// TIA Portal project "Örnek Asansör" (V16)

(* hardware
DEVICE "S71500/ET200MP station_1"  S7-1500 station
   slot 0: "Rail_0"  Rack  6ES7 590-1***0-0AA0
   slot 1: "PLC_1"  CPU 1517-3 PN/DP  6ES7 517-3AP00-0AB0  V2.8
      slot 3: "CPU display_1"  6ES7591-1BA00-0AA0
      slot 32768: "PROFINET interface_1"  X1
         slot 32769: "Port_1"  X1 P1
         slot 32770: "Port_2"  X1 P2
      slot 33024: "PROFINET interface_2"  X2
         slot 33025: "Port_1"  X2 P1
      slot 33280: "DP interface_1"  X3
      slot 34817: "Virtual CP interface port_1"  Virtual CP interface port  Virtual CP interface port
DEVICE "HMI_1"  TP1500 Comfort
   slot 0: "HMI_1"  TP1500 Comfort  6AV2 124-0QC02-0AX1  16.0.0.0
   slot 1: "HMI_RT_1"  TP1500 Comfort  6AV2 124-0QC02-0AX1  16.0.0.0
   slot 5: "HMI_1.IE_CP_1"  PROFINET Interface  16.0.0.0
      slot 1: "PROFINET Interface_1"  PROFINET Interface
         slot 1: "Port_1"  Port
         slot 2: "Port_2"  Port
   slot 6: "HMI_1.IE_CP_2"  PROFINET Interface  16.0.0.0
      slot 1: "PROFINET Interface_GBit"  PROFINET Interface
         slot 1: "Port_1"  Port
   slot 7: "HMI_1.MPI/DP_CP_1"  MPI/DP Interface  16.0.0.0
*)

// ===== PLC "PLC_1"  CPU 1517-3 PN/DP =====

VAR_GLOBAL   // PLC tag table "Default tag table"
   "Asansor0Katta" AT %M10.0 : Bool;
   "Asansor1Katta" AT %M10.1 : Bool;
   "Asansor2Katta" AT %M10.2 : Bool;
   "Asansor3Katta" AT %M10.3 : Bool;
   "0KattanYukarıCag" AT %M11.0 : Bool;
   "1KattanYukarıCag" AT %M11.1 : Bool;
   "1KattanAsagıCag" AT %M11.2 : Bool;
   "2KattanYukarıCag" AT %M11.3 : Bool;
   "2KattanAsagıCag" AT %M11.4 : Bool;
   "3KattanYukarıCag" AT %M11.5 : Bool;
   "3KattanAsagıCag" AT %M11.6 : Bool;
   "0KataGit" AT %M12.0 : Bool;
   "1KataGit" AT %M12.1 : Bool;
   "2KataGit" AT %M12.2 : Bool;
   "3KataGit" AT %M12.3 : Bool;
   "IsıkBariyeriGüvenli" AT %M13.0 : Bool;
   "KapıAcık" AT %M14.0 : Bool;
   "KapıKapalı" AT %M14.1 : Bool;
   "AsansorYukarı" AT %M20.0 : Bool;
   "AsansorAsagı" AT %M20.1 : Bool;
   "KapıKapatKat0" AT %M21.0 : Bool;
   "KapıAcKat0" AT %M21.1 : Bool;
   "KapıKapatKat1" AT %M22.0 : Bool;
   "KapıAcKat1" AT %M22.1 : Bool;
   "KapaKapatKat2" AT %M23.0 : Bool;
   "KapıAcKat2" AT %M23.1 : Bool;
   "KapıKapatKat3" AT %M24.0 : Bool;
   "KapıAcat3" AT %M24.1 : Bool;
   "P_TRIG1" AT %M0.0 : Bool;
   "P_TRIG2" AT %M0.1 : Bool;
   "P_TRIG3" AT %M0.2 : Bool;
   "P_TRIG4" AT %M0.3 : Bool;
   "P_TRIG5" AT %M0.4 : Bool;
   "P_TRIG6" AT %M1.0 : Bool;
   "P_TRIG7" AT %M1.1 : Bool;
   "P_TRIG8" AT %M1.2 : Bool;
   "P_TRIG9" AT %M0.5 : Bool;
   "P_TRIG10" AT %M0.6 : Bool;
   "P_TRIG11" AT %M0.7 : Bool;
   "P_TRIG12" AT %M1.3 : Bool;
   "P_TRIG13" AT %M1.4 : Bool;
   "IsıkBariyeriGüvenlik" AT %M1.5 : Bool;
   "P_TRIG14" AT %M1.6 : Bool;
   "P_TRIG15" AT %M1.7 : Bool;
   "P_TRIG16" AT %M2.0 : Bool;
   "P_TRIG17" AT %M2.1 : Bool;
   "P_TRIG18" AT %M2.2 : Bool;
   "P_TRIG19" AT %M2.3 : Bool;
   "P_TRIG20" AT %M2.4 : Bool;
   "P_TRIG21" AT %M2.5 : Bool;
   "P_TRIG22" AT %M2.6 : Bool;
   "P_TRIG23" AT %M2.7 : Bool;
   "P_TRIG24" AT %M3.0 : Bool;
   "P_TRIG25" AT %M3.1 : Bool;
   "P_TRIG26" AT %M3.2 : Bool;
   "P_TRIG27" AT %M3.3 : Bool;
   "P_TRIG28" AT %M3.4 : Bool;
   "P_TRIG29" AT %M3.5 : Bool;
   "deneme" AT %M3.6 : Bool;
   "P_TRIG30" AT %M3.7 : Bool;
   "P_TRIG31" AT %M4.0 : Bool;
   "P_TRIG32" AT %M4.1 : Bool;
   "P_TRIG33" AT %M4.2 : Bool;
   "P_TRIG34" AT %M4.3 : Bool;
   "P_TRIG35" AT %M4.4 : Bool;
   "P_TRIG36" AT %M4.5 : Bool;
   "P_TRIG37" AT %M4.6 : Bool;
   "P_TRIG38" AT %M4.7 : Bool;
   "P_TRIG39" AT %M5.0 : Bool;
   "P_TRIG40" AT %M5.1 : Bool;
   "P_TRIG42" AT %M5.2 : Bool;
   "P_TRIG43" AT %M5.3 : Bool;
   "P_TRIG41" AT %M5.4 : Bool;
   "P_TRIG44" AT %M5.5 : Bool;
   "P_TRIG47" AT %M5.6 : Bool;
   "P_TRIG48" AT %M5.7 : Bool;
   "P_TRIG46" AT %M6.0 : Bool;
   "P_TRIG45" AT %M6.1 : Bool;
   "P_TRIG67" AT %M6.2 : Bool;
   "P_TRIG68" AT %M6.3 : Bool;
   "P_TRIG69" AT %M6.4 : Bool;
   "1k" AT %M6.5 : Bool;
   "P_TRIG70" AT %M6.6 : Bool;
   "2k" AT %M6.7 : Bool;
   "3k" AT %M7.0 : Bool;
   "d1" AT %M7.1 : Bool;
   "P-TRIG671" AT %M7.2 : Bool;
   "d2" AT %M7.3 : Bool;
   "P_TRIG72" AT %M7.4 : Bool;
   "d3" AT %M7.5 : Bool;
   "P_TRIG73" AT %M7.6 : Bool;
   "P_TRIG74" AT %M7.7 : Bool;
   "P_TRIG75" AT %M8.0 : Bool;
   "P_TRIG76" AT %M8.1 : Bool;
   "P_TRIG77" AT %M8.2 : Bool;
   "P_TRIG78" AT %M8.3 : Bool;
   "P_TRIG79" AT %M8.4 : Bool;
   "P_TRIG80" AT %M8.5 : Bool;
   "P_TRIG81" AT %M8.6 : Bool;
   "P_TRIG82" AT %M8.7 : Bool;
   "P_TRIG84" AT %M9.0 : Bool;
   "P_TRIG85" AT %M9.1 : Bool;
   "P_TRIG100" AT %M80.0 : Bool;
   "11k" AT %M80.1 : Bool;
   "22k" AT %M9.2 : Bool;
   "Yukarı" AT %M9.3 : Bool;
   "P_TRIG101" AT %M9.4 : Bool;
   "P_TRIG102" AT %M9.5 : Bool;
   "33k" AT %M9.6 : Bool;
   "d11" AT %M9.7 : Bool;
   "P_TRIG103" AT %M10.4 : Bool;
   "P_TRIG105" AT %M10.5 : Bool;
   "P_TRIG104" AT %M10.6 : Bool;
   "d22" AT %M10.7 : Bool;
   "P_TRIG106" AT %M11.7 : Bool;
   "P_TRIG107" AT %M12.4 : Bool;
   "d33" AT %M12.5 : Bool;
   "P_TRIG108" AT %M12.6 : Bool;
   "P_TRIG109" AT %M12.7 : Bool;
   "P_TRIG110" AT %M13.1 : Bool;
   "P_TRIG111" AT %M13.2 : Bool;
   "P_TRIG112" AT %M13.3 : Bool;
   "P_TRIG114" AT %M13.4 : Bool;
   "P_TRIG113" AT %M13.5 : Bool;
   "111k" AT %M13.6 : Bool;
   "222k" AT %M13.7 : Bool;
   "333k" AT %M14.2 : Bool;
   "P_TRIG115" AT %M14.3 : Bool;
   "P_TRIG116" AT %M14.4 : Bool;
   "P_TRIG117" AT %M14.5 : Bool;
   "P_TRIG118" AT %M14.6 : Bool;
   "d111" AT %M14.7 : Bool;
   "P_TRIG119" AT %M15.0 : Bool;
   "P_TRIG120" AT %M15.1 : Bool;
   "d222" AT %M15.2 : Bool;
   "d333" AT %M15.3 : Bool;
   "P_TRIG121" AT %M15.4 : Bool;
   "P_TRIG122" AT %M15.5 : Bool;
   "P_TRIG123" AT %M15.6 : Bool;
   "P_TRIG124" AT %M15.7 : Bool;
   "P_TRIG128" AT %M16.0 : Bool;
   "P_TRIG127" AT %M16.1 : Bool;
   "P_TRIG126" AT %M16.2 : Bool;
   "P_TRIG125" AT %M16.3 : Bool;
   "P_TRIG129" AT %M16.4 : Bool;
   "P_TRIG130" AT %M16.5 : Bool;
   "1111k" AT %M16.6 : Bool;
   "P_TRIG131" AT %M16.7 : Bool;
   "3333k" AT %M17.0 : Bool;
   "2222k" AT %M17.1 : Bool;
   "P_TRIG132" AT %M17.2 : Bool;
   "P_TRIG133" AT %M17.3 : Bool;
   "P_TRIG134" AT %M17.4 : Bool;
   "P_TRIG135" AT %M17.5 : Bool;
   "P_TRIG136" AT %M17.6 : Bool;
   "P_TRIG137" AT %M17.7 : Bool;
   "P_TRIG138" AT %M18.0 : Bool;
   "P_TRIG139" AT %M18.1 : Bool;
   "P_TRIG140" AT %M18.2 : Bool;
END_VAR

// folder: System blocks/Program resources

DATA_BLOCK "IEC_Timer_0_DB"   // DB1
{ S7_Optimized_Access := 'TRUE' }
AUTHOR : Simatic
FAMILY : IEC
NAME : IEC_TMR
VERSION : 1.0
// stored: InstanceOfName IEC_TIMER
"IEC_TIMER"
BEGIN
END_DATA_BLOCK

DATA_BLOCK "IEC_Timer_0_DB_1"   // DB2
{ S7_Optimized_Access := 'TRUE' }
AUTHOR : Simatic
FAMILY : IEC
NAME : IEC_TMR
VERSION : 1.0
// stored: InstanceOfName IEC_TIMER
"IEC_TIMER"
BEGIN
END_DATA_BLOCK

DATA_BLOCK "IEC_Timer_0_DB_2"   // DB3
{ S7_Optimized_Access := 'TRUE' }
AUTHOR : Simatic
FAMILY : IEC
NAME : IEC_TMR
VERSION : 1.0
// stored: InstanceOfName IEC_TIMER
"IEC_TIMER"
BEGIN
END_DATA_BLOCK

DATA_BLOCK "IEC_Timer_0_DB_3"   // DB4
{ S7_Optimized_Access := 'TRUE' }
AUTHOR : Simatic
FAMILY : IEC
NAME : IEC_TMR
VERSION : 1.0
// stored: InstanceOfName IEC_TIMER
"IEC_TIMER"
BEGIN
END_DATA_BLOCK

// folder: (top level)

ORGANIZATION_BLOCK "Main"   // OB1, LAD, ProgramCycle
TITLE = "Main Program Sweep (Cycle)"
{ S7_Optimized_Access := 'TRUE' }
VERSION : 0.1
   VAR_INPUT
      Initial_Call : Bool;   // Initial call of this OB
      Remanence : Bool;   // =True, if remanent data are available
   END_VAR
   VAR_TEMP
      P_TRIG83 : Bool;
   END_VAR
   VAR_TEMP   // added for the SCL form of the ladder/FBD networks
      _w1 : Bool;
      _w2 : Bool;
      _w3 : Bool;
      _w4 : Bool;
      _w5 : Bool;
      _w6 : Bool;
      _w7 : Bool;
      _w8 : Bool;
      _w9 : Bool;
      _w10 : Bool;
      _w11 : Bool;
      _w12 : Bool;
      _w13 : Bool;
      _w14 : Bool;
      _w15 : Bool;
      _w16 : Bool;
      _w17 : Bool;
      _w18 : Bool;
      _w19 : Bool;
      _w20 : Bool;
      _w21 : Bool;
      _w22 : Bool;
      _w23 : Bool;
      _w24 : Bool;
      _w25 : Bool;
      _w26 : Bool;
      _w27 : Bool;
      _w28 : Bool;
      _w29 : Bool;
   END_VAR
BEGIN

REGION Network 1: 0 dan 1-2-3 Çıkış
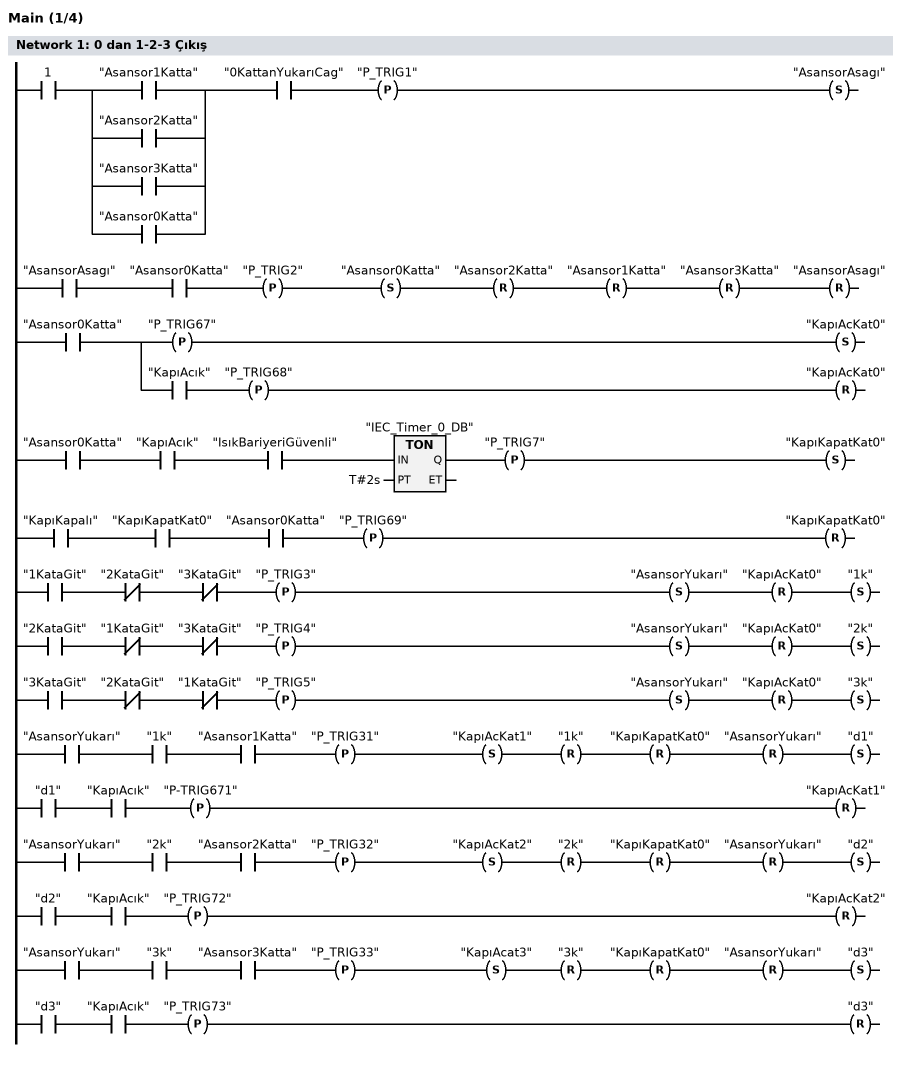
   #_w1 := 1 AND ("Asansor1Katta" OR "Asansor2Katta" OR "Asansor3Katta" OR "Asansor0Katta") AND "0KattanYukarıCag";
   #_w2 := #_w1 AND NOT "P_TRIG1";   // rising edge
   "P_TRIG1" := #_w1;
   IF #_w2 THEN "AsansorAsagı" := TRUE; END_IF;
   #_w3 := "AsansorAsagı" AND "Asansor0Katta";
   #_w4 := #_w3 AND NOT "P_TRIG2";   // rising edge
   "P_TRIG2" := #_w3;
   IF #_w4 THEN
       "Asansor0Katta" := TRUE;
       "Asansor2Katta" := FALSE;
       "Asansor1Katta" := FALSE;
       "Asansor3Katta" := FALSE;
       "AsansorAsagı" := FALSE;
   END_IF;
   #_w5 := "Asansor0Katta" AND NOT "P_TRIG67";   // rising edge
   "P_TRIG67" := "Asansor0Katta";
   IF #_w5 THEN "KapıAcKat0" := TRUE; END_IF;
   #_w6 := "Asansor0Katta" AND "KapıAcık";
   #_w7 := #_w6 AND NOT "P_TRIG68";   // rising edge
   "P_TRIG68" := #_w6;
   IF #_w7 THEN "KapıAcKat0" := FALSE; END_IF;
   "IEC_Timer_0_DB".TON(IN := "Asansor0Katta" AND "KapıAcık" AND "IsıkBariyeriGüvenli", PT := T#2s);
   #_w8 := "IEC_Timer_0_DB".Q AND NOT "P_TRIG7";   // rising edge
   "P_TRIG7" := "IEC_Timer_0_DB".Q;
   IF #_w8 THEN "KapıKapatKat0" := TRUE; END_IF;
   #_w9 := "KapıKapalı" AND "KapıKapatKat0" AND "Asansor0Katta";
   #_w10 := #_w9 AND NOT "P_TRIG69";   // rising edge
   "P_TRIG69" := #_w9;
   IF #_w10 THEN "KapıKapatKat0" := FALSE; END_IF;
   #_w11 := "1KataGit" AND NOT "2KataGit" AND NOT "3KataGit";
   #_w12 := #_w11 AND NOT "P_TRIG3";   // rising edge
   "P_TRIG3" := #_w11;
   IF #_w12 THEN
       "AsansorYukarı" := TRUE;
       "KapıAcKat0" := FALSE;
       "1k" := TRUE;
   END_IF;
   #_w13 := "2KataGit" AND NOT "1KataGit" AND NOT "3KataGit";
   #_w14 := #_w13 AND NOT "P_TRIG4";   // rising edge
   "P_TRIG4" := #_w13;
   IF #_w14 THEN
       "AsansorYukarı" := TRUE;
       "KapıAcKat0" := FALSE;
       "2k" := TRUE;
   END_IF;
   #_w15 := "3KataGit" AND NOT "2KataGit" AND NOT "1KataGit";
   #_w16 := #_w15 AND NOT "P_TRIG5";   // rising edge
   "P_TRIG5" := #_w15;
   IF #_w16 THEN
       "AsansorYukarı" := TRUE;
       "KapıAcKat0" := FALSE;
       "3k" := TRUE;
   END_IF;
   #_w17 := "AsansorYukarı" AND "1k" AND "Asansor1Katta";
   #_w18 := #_w17 AND NOT "P_TRIG31";   // rising edge
   "P_TRIG31" := #_w17;
   IF #_w18 THEN
       "KapıAcKat1" := TRUE;
       "1k" := FALSE;
       "KapıKapatKat0" := FALSE;
       "AsansorYukarı" := FALSE;
       "d1" := TRUE;
   END_IF;
   #_w19 := "d1" AND "KapıAcık";
   #_w20 := #_w19 AND NOT "P-TRIG671";   // rising edge
   "P-TRIG671" := #_w19;
   IF #_w20 THEN "KapıAcKat1" := FALSE; END_IF;
   #_w21 := "AsansorYukarı" AND "2k" AND "Asansor2Katta";
   #_w22 := #_w21 AND NOT "P_TRIG32";   // rising edge
   "P_TRIG32" := #_w21;
   IF #_w22 THEN
       "KapıAcKat2" := TRUE;
       "2k" := FALSE;
       "KapıKapatKat0" := FALSE;
       "AsansorYukarı" := FALSE;
       "d2" := TRUE;
   END_IF;
   #_w23 := "d2" AND "KapıAcık";
   #_w24 := #_w23 AND NOT "P_TRIG72";   // rising edge
   "P_TRIG72" := #_w23;
   IF #_w24 THEN "KapıAcKat2" := FALSE; END_IF;
   #_w25 := "AsansorYukarı" AND "3k" AND "Asansor3Katta";
   #_w26 := #_w25 AND NOT "P_TRIG33";   // rising edge
   "P_TRIG33" := #_w25;
   IF #_w26 THEN
       "KapıAcat3" := TRUE;
       "3k" := FALSE;
       "KapıKapatKat0" := FALSE;
       "AsansorYukarı" := FALSE;
       "d3" := TRUE;
   END_IF;
   #_w27 := "d3" AND "KapıAcık";
   #_w28 := #_w27 AND NOT "P_TRIG73";   // rising edge
   "P_TRIG73" := #_w27;
   IF #_w28 THEN "d3" := FALSE; END_IF;
END_REGION

REGION Network 2: 1 den 2-3 çıkış ya da 0 a iniş
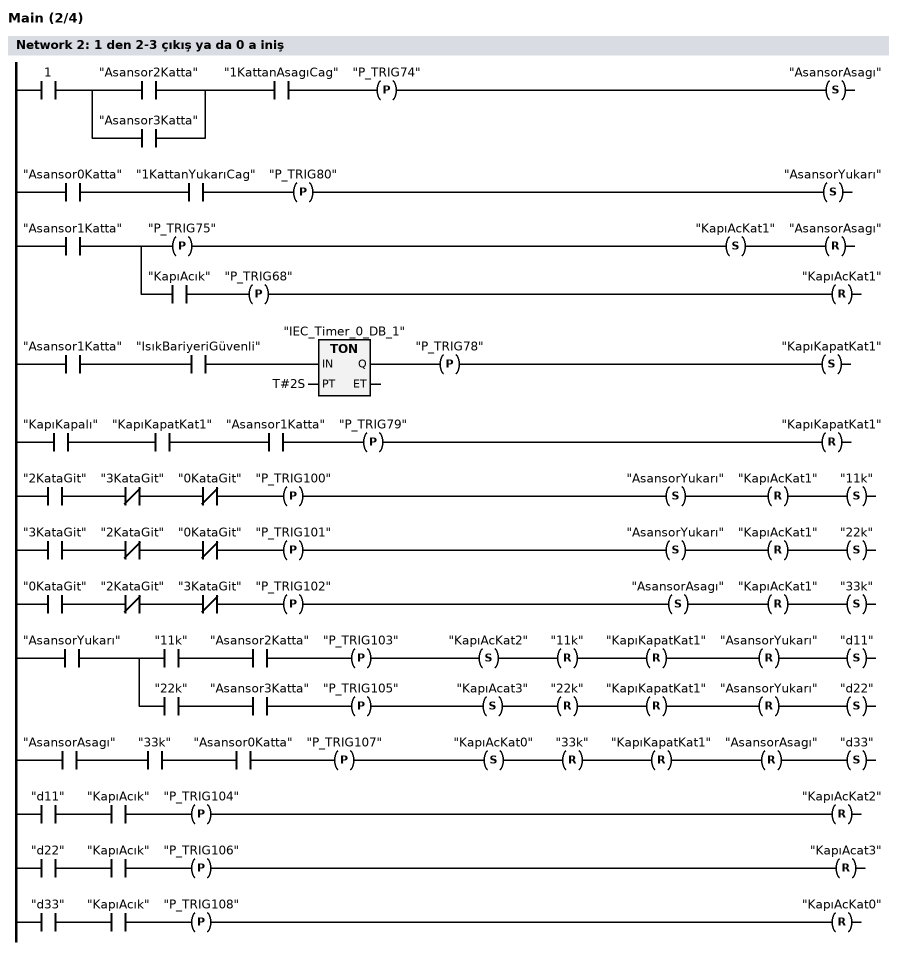
   #_w1 := 1 AND ("Asansor2Katta" OR "Asansor3Katta") AND "1KattanAsagıCag";
   #_w2 := #_w1 AND NOT "P_TRIG74";   // rising edge
   "P_TRIG74" := #_w1;
   IF #_w2 THEN "AsansorAsagı" := TRUE; END_IF;
   #_w3 := "Asansor0Katta" AND "1KattanYukarıCag";
   #_w4 := #_w3 AND NOT "P_TRIG80";   // rising edge
   "P_TRIG80" := #_w3;
   IF #_w4 THEN "AsansorYukarı" := TRUE; END_IF;
   #_w5 := "Asansor1Katta" AND NOT "P_TRIG75";   // rising edge
   "P_TRIG75" := "Asansor1Katta";
   IF #_w5 THEN
       "KapıAcKat1" := TRUE;
       "AsansorAsagı" := FALSE;
   END_IF;
   #_w6 := "Asansor1Katta" AND "KapıAcık";
   #_w7 := #_w6 AND NOT "P_TRIG68";   // rising edge
   "P_TRIG68" := #_w6;
   IF #_w7 THEN "KapıAcKat1" := FALSE; END_IF;
   "IEC_Timer_0_DB_1".TON(IN := "Asansor1Katta" AND "IsıkBariyeriGüvenli", PT := T#2S);
   #_w8 := "IEC_Timer_0_DB_1".Q AND NOT "P_TRIG78";   // rising edge
   "P_TRIG78" := "IEC_Timer_0_DB_1".Q;
   IF #_w8 THEN "KapıKapatKat1" := TRUE; END_IF;
   #_w9 := "KapıKapalı" AND "KapıKapatKat1" AND "Asansor1Katta";
   #_w10 := #_w9 AND NOT "P_TRIG79";   // rising edge
   "P_TRIG79" := #_w9;
   IF #_w10 THEN "KapıKapatKat1" := FALSE; END_IF;
   #_w11 := "2KataGit" AND NOT "3KataGit" AND NOT "0KataGit";
   #_w12 := #_w11 AND NOT "P_TRIG100";   // rising edge
   "P_TRIG100" := #_w11;
   IF #_w12 THEN
       "AsansorYukarı" := TRUE;
       "KapıAcKat1" := FALSE;
       "11k" := TRUE;
   END_IF;
   #_w13 := "3KataGit" AND NOT "2KataGit" AND NOT "0KataGit";
   #_w14 := #_w13 AND NOT "P_TRIG101";   // rising edge
   "P_TRIG101" := #_w13;
   IF #_w14 THEN
       "AsansorYukarı" := TRUE;
       "KapıAcKat1" := FALSE;
       "22k" := TRUE;
   END_IF;
   #_w15 := "0KataGit" AND NOT "2KataGit" AND NOT "3KataGit";
   #_w16 := #_w15 AND NOT "P_TRIG102";   // rising edge
   "P_TRIG102" := #_w15;
   IF #_w16 THEN
       "AsansorAsagı" := TRUE;
       "KapıAcKat1" := FALSE;
       "33k" := TRUE;
   END_IF;
   #_w17 := "AsansorYukarı" AND "11k" AND "Asansor2Katta";
   #_w18 := #_w17 AND NOT "P_TRIG103";   // rising edge
   "P_TRIG103" := #_w17;
   IF #_w18 THEN
       "KapıAcKat2" := TRUE;
       "11k" := FALSE;
       "KapıKapatKat1" := FALSE;
   END_IF;
   #_w19 := "AsansorYukarı";
   IF #_w18 THEN
       "AsansorYukarı" := FALSE;
       "d11" := TRUE;
   END_IF;
   #_w20 := #_w19 AND "22k" AND "Asansor3Katta";
   #_w21 := #_w20 AND NOT "P_TRIG105";   // rising edge
   "P_TRIG105" := #_w20;
   IF #_w21 THEN
       "KapıAcat3" := TRUE;
       "22k" := FALSE;
       "KapıKapatKat1" := FALSE;
       "AsansorYukarı" := FALSE;
       "d22" := TRUE;
   END_IF;
   #_w22 := "AsansorAsagı" AND "33k" AND "Asansor0Katta";
   #_w23 := #_w22 AND NOT "P_TRIG107";   // rising edge
   "P_TRIG107" := #_w22;
   IF #_w23 THEN
       "KapıAcKat0" := TRUE;
       "33k" := FALSE;
       "KapıKapatKat1" := FALSE;
       "AsansorAsagı" := FALSE;
       "d33" := TRUE;
   END_IF;
   #_w24 := "d11" AND "KapıAcık";
   #_w25 := #_w24 AND NOT "P_TRIG104";   // rising edge
   "P_TRIG104" := #_w24;
   IF #_w25 THEN "KapıAcKat2" := FALSE; END_IF;
   #_w26 := "d22" AND "KapıAcık";
   #_w27 := #_w26 AND NOT "P_TRIG106";   // rising edge
   "P_TRIG106" := #_w26;
   IF #_w27 THEN "KapıAcat3" := FALSE; END_IF;
   #_w28 := "d33" AND "KapıAcık";
   #_w29 := #_w28 AND NOT "P_TRIG108";   // rising edge
   "P_TRIG108" := #_w28;
   IF #_w29 THEN "KapıAcKat0" := FALSE; END_IF;
END_REGION

REGION Network 3: 2 den 3 e çıkış ya da 1 ve 0 a iniş
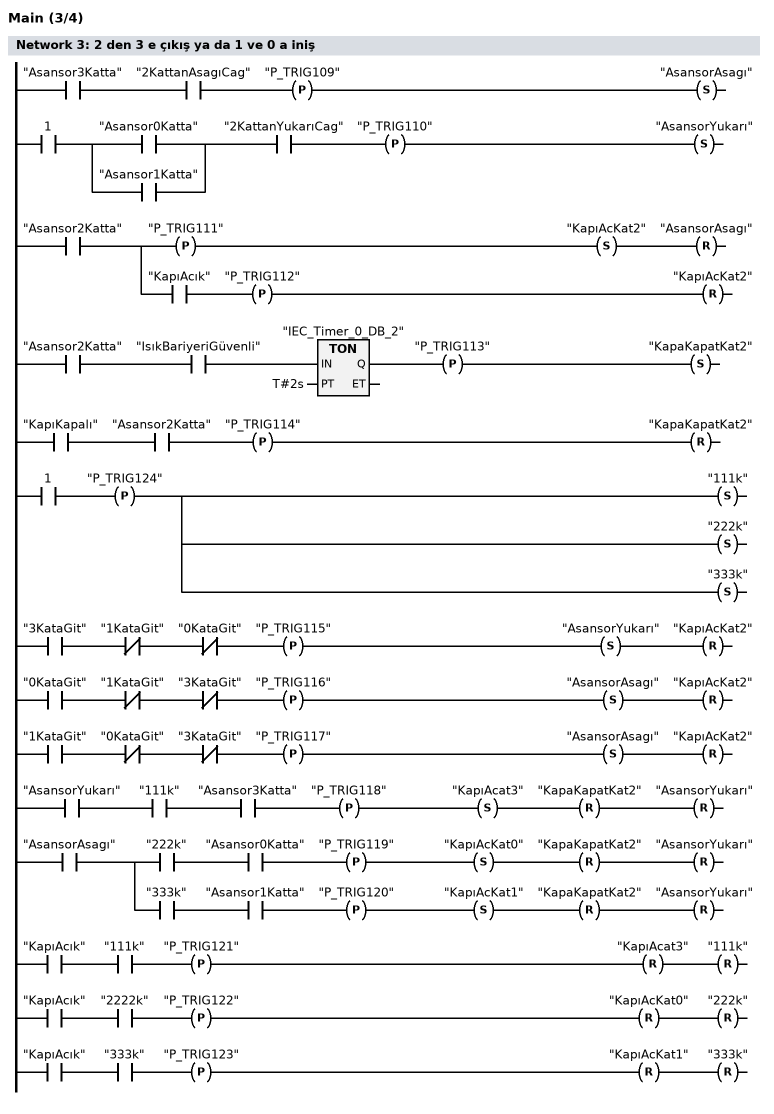
   // no checked SCL form for this network; see the picture
END_REGION

REGION Network 4: 3 . kattan 0 1 2 inme
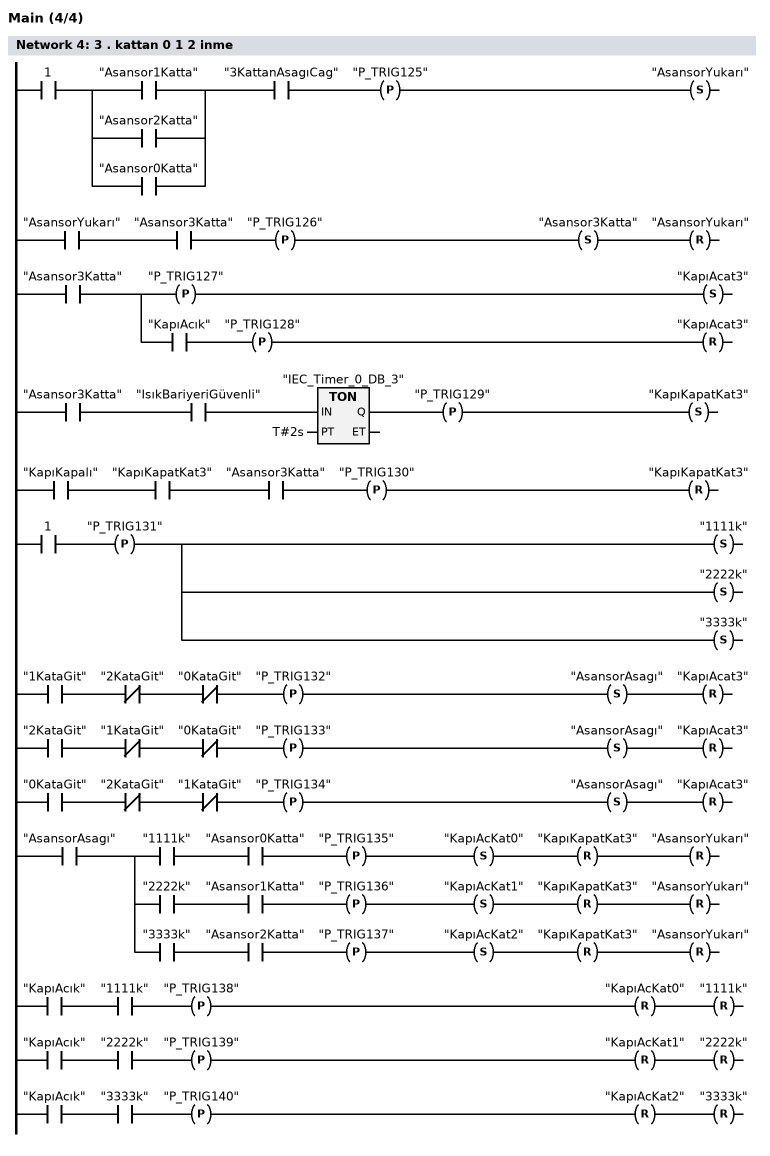
   // no checked SCL form for this network; see the picture
END_REGION
END_ORGANIZATION_BLOCK

(* ===== HMI "HMI_RT_1" =====
system functions are stored by id; their names below are inferred from use
connection "HMI_Connection_1": ETHERNET, S7_1500_OMS

HMI tags "Default tag table"
   "Tag_ScreenNumber" : UInt, internal
   "3KataGit" : Bool = PLC 3KataGit AT %M12.3, 1 s
   "2KataGit" : Bool = PLC 2KataGit AT %M12.2, 1 s
   "1KataGit" : Bool = PLC 1KataGit AT %M12.1, 1 s
   "0KataGit" : Bool = PLC 0KataGit AT %M12.0, 1 s
   "0KattanYukarıCag" : Bool = PLC 0KattanYukarıCag AT %M11.0, 1 s
   "1KattanYukarıCag" : Bool = PLC 1KattanYukarıCag AT %M11.1, 1 s
   "1KattanAsagıCag" : Bool = PLC 1KattanAsagıCag AT %M11.2, 1 s
   "2KattanYukarıCag" : Bool = PLC 2KattanYukarıCag AT %M11.3, 1 s
   "2KattanAsagıCag" : Bool = PLC 2KattanAsagıCag AT %M11.4, 1 s
   "3KattanAsagıCag" : Bool = PLC 3KattanAsagıCag AT %M11.6, 1 s
   "Asansor0Katta" : Bool = PLC Asansor0Katta AT %M10.0, 1 s
   "Asansor1Katta" : Bool = PLC Asansor1Katta AT %M10.1, 1 s
   "Asansor3Katta" : Bool = PLC Asansor3Katta AT %M10.3, 1 s
   "Asansor2Katta" : Bool = PLC Asansor2Katta AT %M10.2, 1 s
   "KapıAcık" : Bool = PLC KapıAcık AT %M14.0, 1 s
   "KapıKapalı" : Bool = PLC KapıKapalı AT %M14.1, 1 s
   "AsansorYukarı" : Bool = PLC AsansorYukarı AT %M20.0, 1 s
   "AsansorAsagı" : Bool = PLC AsansorAsagı AT %M20.1, 1 s
   "IsıkBariyeriGüvenli" : Bool = PLC IsıkBariyeriGüvenli AT %M13.0, 1 s
   "KapıKapalıKat0" : Bool = PLC KapıKapatKat0 AT %M21.0, 1 s
   "KapıAcıkKat0" : Bool = PLC KapıAcKat0 AT %M21.1, 1 s
   "KapıKapalıKat1" : Bool = PLC KapıKapatKat1 AT %M22.0, 1 s
   "KapıAcıkKat1" : Bool = PLC KapıAcKat1 AT %M22.1, 1 s
   "KapaKapalıKat2" : Bool = PLC KapaKapatKat2 AT %M23.0, 1 s
   "KapıAcıkKat2" : Bool = PLC KapıAcKat2 AT %M23.1, 1 s
   "KapıKapalıKat3" : Bool = PLC KapıKapatKat3 AT %M24.0, 1 s
   "KapıAcıkKat3" : Bool = PLC KapıAcat3 AT %M24.1, 1 s

screen "Root screen" 1280x740, template "Template_1"
   on GenerateScreen: SetTag("Tag_ScreenNumber", 1)
   GraphicIOField "Graphic I/O field_1" at 734,50 size 328x410
   GraphicIOField "Graphic I/O field_2" at 740,55 size 191x400
   Button "Button_1" at 953,62 size 96x32; TextOff '3.Kat'
      on Press: function_b14e0dd5("3KataGit", 0)
   Button "Button_2" at 956,132 size 96x32; TextOff '2.Kat'
      on Press: function_b14e0dd5("2KataGit", 0)
   Button "Button_3" at 956,208 size 96x32; TextOff '1.Kat'
      on Press: function_b14e0dd5("1KataGit", 0)
   Button "Button_4" at 953,288 size 96x32; TextOff '0.Kat'
      on Press: function_b14e0dd5("0KataGit", 0)
   Button "Button_5" at 40,31 size 109x32; TextOff '0.Kat Up'
      on Press: function_b14e0dd5("0KattanYukarıCag", 0)
   Button "Button_6" at 40,75 size 109x32; TextOff '1.Kat Up'
      on Press: function_b14e0dd5("1KattanYukarıCag", 0)
   Button "Button_7" at 39,115 size 110x32; TextOff '2.Kat Up'
      on Press: function_b14e0dd5("2KattanYukarıCag", 0)
   Button "Button_8" at 39,163 size 109x32; TextOff '3.Kat Down'
      on Press: function_b14e0dd5("3KattanAsagıCag", 0)
   Button "Button_9" at 187,73 size 108x32; TextOff '1.Kat Down'
      on Press: function_b14e0dd5("1KattanAsagıCag", 0)
   Button "Button_10" at 187,113 size 108x32; TextOff '2.Kat Down'
      on Press: function_b14e0dd5("2KattanAsagıCag", 0)
   Button "Button_11" at 3,256 size 244x32; TextOff 'Asansör 0. Katta Sensor'
      on Press: InvertBit("Asansor0Katta")
   Button "Button_12" at 0,306 size 256x32; TextOff 'Asansör 1. Katta Sensor'
      on Press: SetBit("Asansor1Katta")
   Button "Button_13" at 3,367 size 239x32; TextOff 'Asansör 2. Katta'
      on Press: InvertBit("Asansor2Katta")
   Button "Button_14" at 3,428 size 260x32; TextOff 'Asansör 3. Katta'
      on Press: InvertBit("Asansor3Katta")
   Button "Button_15" at 38,471 size 102x32; TextOff 'Kapı Açık'
      on Press: InvertBit("KapıAcık")
   Button "Button_16" at 41,531 size 100x32; TextOff 'Kapı Kapalı'
      on Press: InvertBit("KapıKapalı")
      Appearance <- "KapıKapalı"
   Circle "Circle_1" at 271,475 size 48x48
      Appearance <- "KapıAcık"
   Circle "Circle_2" at 271,531 size 48x48
      Appearance <- "KapıKapalı"
   TextField "Text field_1" at 377,27 size 154x25; Text 'Asansör Yukarı:'
   Circle "Circle_3" at 538,8 size 48x48
      Appearance <- "AsansorYukarı"
   TextField "Text field_2" at 377,66 size 146x25; Text 'Asansör Aşağı:'
   Circle "Circle_4" at 538,56 size 48x48
      Appearance <- "AsansorAsagı"
   Button "Button_17" at 367,131 size 142x32; TextOff 'Işık-Güvenlik'
      on Press: InvertBit("IsıkBariyeriGüvenli")
   Circle "Circle_5" at 543,120 size 48x48
      Appearance <- "IsıkBariyeriGüvenli"
   Circle "Circle_6" at 271,240 size 48x48
      Appearance <- "Asansor0Katta"
   Circle "Circle_7" at 273,290 size 48x48
      Appearance <- "Asansor1Katta"
   Circle "Circle_8" at 273,345 size 48x48
      Appearance <- "Asansor2Katta"
   Circle "Circle_9" at 271,404 size 48x48
      Appearance <- "Asansor3Katta"
   TextField "Text field_3" at 369,240 size 164x25; Text 'Kapı Kapat 0.Kat'
   Circle "Circle_10" at 545,231 size 48x48
      Appearance <- "KapıKapalıKat0"
   TextField "Text field_4" at 367,296 size 132x25; Text 'Kapı Aç 0.Kat'
   Circle "Circle_11" at 543,287 size 48x48
      Appearance <- "KapıAcıkKat0"
   TextField "Text field_5" at 365,352 size 164x25; Text 'Kapı Kapat 1.Kat'
   Circle "Circle_12" at 541,343 size 48x48
      Appearance <- "KapıKapalıKat1"
   TextField "Text field_6" at 363,408 size 132x25; Text 'Kapı Aç 1.Kat'
   Circle "Circle_13" at 539,399 size 48x48
      Appearance <- "KapıAcıkKat1"
   TextField "Text field_7" at 361,464 size 164x25; Text 'Kapı Kapat 2.Kat'
   Circle "Circle_14" at 537,455 size 48x48
      Appearance <- "KapaKapalıKat2"
   TextField "Text field_8" at 359,520 size 132x25; Text 'Kapı Aç 2.Kat'
   Circle "Circle_15" at 535,511 size 48x48
      Appearance <- "KapıAcıkKat2"
   TextField "Text field_9" at 357,576 size 164x25; Text 'Kapı Kapat 3.Kat'
   Circle "Circle_16" at 533,567 size 48x48
      Appearance <- "KapıKapalıKat3"
   TextField "Text field_10" at 355,632 size 132x25; Text 'Kapı Aç 3.Kat'
   Circle "Circle_17" at 531,623 size 48x48
      Appearance <- "KapıAcıkKat3"

Template "Template_1" 1280x740
   Button "Exit" at 1200,679 size 78x59; TextOff 'Exit'; PictureOff "ExitRuntime_TP1500_Comfort_V2_TR"; PictureOn "ExitRuntime_TP1500_Comfort_V2_TR"
      on Release: StopRuntime(0)
   Button "Template_Button" at 1120,679 size 78x59; TextOff 'Text'
   Button "Template_Button_1" at 1040,679 size 78x59; TextOff 'Text'
   Button "Template_Button_2" at 960,679 size 78x59; TextOff 'Text'
   Button "Template_Button_3" at 880,679 size 78x59; TextOff 'Text'
   Button "Template_Button_4" at 800,679 size 78x59; TextOff 'Text'
   Button "Template_Button_5" at 720,679 size 78x59; TextOff 'Text'
   Button "Template_Button_6" at 640,679 size 78x59; TextOff 'Text'
   Button "Template_Button_7" at 561,679 size 78x59; TextOff 'Text'
   Button "Template_Button_8" at 481,679 size 78x59; TextOff 'Text'
   Button "Template_Button_9" at 401,679 size 78x59; TextOff 'Text'
   Button "Template_Button_10" at 321,679 size 78x59; TextOff 'Text'
   Button "Template_Button_11" at 241,679 size 78x59; TextOff 'Text'
   Button "Template_Button_12" at 161,679 size 78x59; TextOff 'Text'
   Button "Template_Button_13" at 81,679 size 78x59; TextOff 'Text'
   Button "Start screen" at 1,679 size 78x59; TextOff 'Start screen'; PictureOff "NavigateHome_TP1500_Comfort_V2_TR"; PictureOn "NavigateHome_TP1500_Comfort_V2_TR"
      on Release: ActivateScreen("Root screen", 0)
*)